// TIA Portal V20 export
TYPE "typeSequenceControlNodeJobInterface"
// stored: Namespace Unit1.Em0
   STRUCT
      commands { ExternalWritable := 'False'} : "unit1.em0.typeSequenceControlNodeJobInterfaceCommands";
      monitoring { ExternalWritable := 'False'} : "unit1.em0.typeSequenceControlNodeJobInterfaceMonitoring";
   END_STRUCT;
END_TYPE
